// TwinCAT 3 PLC project LabExercise
// ProgramVersion: 3.1.4023.0
// libraries:
//   Tc2_NCI, * (Beckhoff Automation GmbH)
//   Tc2_Standard, * (Beckhoff Automation GmbH)
//   Tc2_System, * (Beckhoff Automation GmbH)
//   Tc3_Module, * (Beckhoff Automation GmbH)
//   VisuDialogs, * (System)
// project tree:
//   Comissioning/Function blocks/ FB_ModifyAutomaticControlSettings.TcPOU (not stored)
//   Comissioning/GVLs/ G_Commissioning.TcGVL (not stored)
//   Comissioning/Struct/ ST_AutomaticControlSettings.TcDUT (not stored), ST_ClosedLoopControlSettings.TcDUT (not stored), ST_MotionReferenceGeneratorSettings.TcDUT (not stored), ST_OpenLoopControlSettings.TcDUT (not stored)
//   ControlBox/Interfaces/ I_ControlBox.TcIO (not stored)
//   ControlBox/Function blocks/ FB_ControlBox.TcPOU, FB_RealControlBox.TcPOU (not stored), FB_VirtualControlBox.TcPOU (not stored)
//   CraneControl/Function blocks/Sub blocks/ FB_ActiveDamping.TcPOU (not stored), FB_Clock.TcPOU (not stored), FB_ClosedLoopControl.TcPOU (not stored), FB_Joystick.TcPOU (not stored), FB_MotionReferenceGenerator_limit.TcPOU (not stored), FB_OpenLoopControl.TcPOU (not stored), FB_ResetIntegralController.TcPOU (not stored), FB_Status.TcPOU (not stored)
//   CraneControl/Enums/ E_Mode.TcDUT (not stored), E_Status.TcDUT (not stored)
//   CraneControl/Function blocks/Main blocks/ FB_AutomaticControl.TcPOU (not stored), FB_ManualControl.TcPOU (not stored)
//   CraneControl/Functions/ F_BarToEng.TcPOU (not stored), F_LminToEng.TcPOU (not stored), F_RadToDeg.TcPOU (not stored)
//   CraneControl/GVLs/ G_Parameters.TcGVL (not stored), G_Work.TcGVL
//   CraneControl/Struct/ ST_ActiveDamping.TcDUT (not stored), ST_Parameters.TcDUT (not stored)
//   / GlobalTextList.TcGTLO (not stored), PlcTask.TcTTO (not stored), Simulator.TcTTO (not stored), Visualization Manager.TcVMO (not stored)
//   HMI/ HMI.TcVIS
//   HMI/Sub/ CommissioningHMI.TcVIS (not stored), VirtualControlBox.TcVIS (not stored)
//   Inputs/ FB_JoystickInputScaling.TcPOU (not stored), FB_PositionInputScaling.TcPOU (not stored), FB_PressureInputScaling.TcPOU (not stored), G_Inputs.TcGVL (not stored), G_Sensors.TcGVL (not stored)
//   Inputs/Struct/ ST_AnalogInput.TcDUT (not stored), ST_AnalogInputStatus.TcDUT (not stored)
//   Internship/ F_PressureSensorInToBar.TcPOU (not stored), V2Q2u.TcPOU
//   Outputs/ FB_ValveOutput.TcPOU (not stored), G_Outputs.TcGVL (not stored)
//   Outputs/Struct/ ST_pValveDeadBand.TcDUT (not stored), ST_ValveOutput.TcDUT (not stored)
//   ControlBox/GVLs/ G_VirtualControlBox.TcGVL (not stored)
//   Programs/ MAIN.TcPOU, P_Commissioning.TcPOU (not stored), P_ControlBox.TcPOU (not stored), P_CraneControl.TcPOU, P_Inputs.TcPOU (not stored), P_OutputNonCompensated.TcPOU, P_Outputs.TcPOU (not stored), P_Simulator.TcPOU (not stored)
//   Simulator/ FB_CraneSimulator.TcPOU, G_Simulator.TcGVL (not stored)
// real-time tasks:
//   TASK PlcTask: cycle T#1ms, priority 20, ADS port 350
//   TASK Simulator: cycle T#100us, priority 1, ADS port 351
// I/O:
//   DEVICE PLC (EtherCAT) (disabled), AmsNetId 10.229.3.117.2.1
//     PLC Rack (EK1200) [EK1200-5000 EtherCAT Power supply (2A E-Bus)]
//       DI (EL1008) [EL1008 8Ch. Dig. Input 24V, 3ms]
//       DO (EL2008) [EL2008 8Ch. Dig. Output 24V, 0.5A]
//       End Cap 4 (EL9011) [EL9011 End Terminal]
//   DEVICE RIO (EtherCAT) (disabled), AmsNetId 10.229.3.117.5.1
//     RIO (EK1100) [EK1100 EtherCAT Coupler (2A E-Bus)]
//       DI (EL1008) [EL1008 8Ch. Dig. Input 24V, 3ms]
//       DO (EL2008) [EL2008 8Ch. Dig. Output 24V, 0.5A]
//       AI1 (EL3068) [EL3068 8Ch. Ana. Input 0-10V]
//       AI2 (EL3068) [EL3068 8Ch. Ana. Input 0-10V]
//       AI3 (EL3174) [EL3174 4Ch. Ana. Input +/-10V Diff., +/-20mA SingleEnded, 16 Bit]
//       AO (EL4104) [EL4104 4Ch. Ana. Output 0-10V, 16bit]
//       End Cap (EL9011) [EL9011 End Terminal]
// variable links:
//   LabExercise/LabExercise Instance <-> PLC (EtherCAT)/PLC Rack (EK1200)/DI (EL1008)
//     PlcTask Inputs/G_Inputs.bTest <-> Channel 1/Input
//   LabExercise/LabExercise Instance <-> PLC (EtherCAT)/PLC Rack (EK1200)/DO (EL2008)
//     PlcTask Outputs/G_Outputs.bTest <-> Channel 1/Output
//   LabExercise/LabExercise Instance <-> RIO (EtherCAT)/RIO (EK1100)/AI1 (EL3068)
//     PlcTask Inputs/G_Inputs.stCylPos.nValue <-> AI Standard Channel 3/Value
//     PlcTask Inputs/G_Inputs.stCylPos.stStatus <-> AI Standard Channel 3/Status
//     PlcTask Inputs/G_Inputs.stJoyX.nValue <-> AI Standard Channel 1/Value
//     PlcTask Inputs/G_Inputs.stJoyX.stStatus <-> AI Standard Channel 1/Status
//     PlcTask Inputs/G_Inputs.stJoyY.nValue <-> AI Standard Channel 2/Value
//     PlcTask Inputs/G_Inputs.stJoyY.stStatus <-> AI Standard Channel 2/Status
//     PlcTask Inputs/G_Inputs.stSpoolPos.nValue <-> AI Standard Channel 4/Value
//     PlcTask Inputs/G_Inputs.stSpoolPos.stStatus <-> AI Standard Channel 4/Status
//   LabExercise/LabExercise Instance <-> RIO (EtherCAT)/RIO (EK1100)/AI2 (EL3068)
//     PlcTask Inputs/G_Inputs.stPressureCompensator.nValue <-> AI Standard Channel 3/Value
//     PlcTask Inputs/G_Inputs.stPressureCompensator.stStatus <-> AI Standard Channel 3/Status
//     PlcTask Inputs/G_Inputs.stPressureLhvSide.nValue <-> AI Standard Channel 5/Value
//     PlcTask Inputs/G_Inputs.stPressureLhvSide.stStatus <-> AI Standard Channel 5/Status
//     PlcTask Inputs/G_Inputs.stPressurePistonSide.nValue <-> AI Standard Channel 4/Value
//     PlcTask Inputs/G_Inputs.stPressurePistonSide.stStatus <-> AI Standard Channel 4/Status
//     PlcTask Inputs/G_Inputs.stPressureReturn.nValue <-> AI Standard Channel 2/Value
//     PlcTask Inputs/G_Inputs.stPressureReturn.stStatus <-> AI Standard Channel 2/Status
//     PlcTask Inputs/G_Inputs.stPressureRodSide.nValue <-> AI Standard Channel 6/Value
//     PlcTask Inputs/G_Inputs.stPressureRodSide.stStatus <-> AI Standard Channel 6/Status
//     PlcTask Inputs/G_Inputs.stPressureSupply.nValue <-> AI Standard Channel 1/Value
//     PlcTask Inputs/G_Inputs.stPressureSupply.stStatus <-> AI Standard Channel 1/Status
//   LabExercise/LabExercise Instance <-> RIO (EtherCAT)/RIO (EK1100)/AI3 (EL3174)
//     PlcTask Inputs/G_Inputs.stFlowReturnSide.nValue <-> AI Standard Channel 1/Value
//     PlcTask Inputs/G_Inputs.stFlowReturnSide.stStatus <-> AI Standard Channel 1/Status
//   LabExercise/LabExercise Instance <-> RIO (EtherCAT)/RIO (EK1100)/AO (EL4104)
//     PlcTask Outputs/G_Outputs.stValveOutput.nValveOutput <-> AO Output Channel 1/Analog output
//   LabExercise/LabExercise Instance <-> RIO (EtherCAT)/RIO (EK1100)/DI (EL1008)
//     PlcTask Inputs/G_Inputs.bAutoModeSelector <-> Channel 1/Input
//     PlcTask Inputs/G_Inputs.bManualModeSelector <-> Channel 2/Input
//     PlcTask Inputs/G_Inputs.bStartButton <-> Channel 3/Input
//     PlcTask Inputs/G_Inputs.bStopButton <-> Channel 4/Input
//   LabExercise/LabExercise Instance <-> RIO (EtherCAT)/RIO (EK1100)/DO (EL2008)
//     PlcTask Outputs/G_Outputs.bGreenLight <-> Channel 1/Output
//     PlcTask Outputs/G_Outputs.bRedLight <-> Channel 2/Output
//     PlcTask Outputs/G_Outputs.stValveOutput.bEnable <-> Channel 3/Output

// ---- CraneControl/GVLs/G_Work.TcGVL
{attribute 'qualified_only'}
VAR_GLOBAL
	eMode 			: E_Mode;
	eStatus 		: E_Status;
	fJoystickY 		: LREAL;
	bFault 			: BOOL;
	bStartButton 	: BOOL;
	bStopButton 	: BOOL;
	fControlOutputNormalized : LREAL;
END_VAR

// ---- ControlBox/Function blocks/FB_ControlBox.TcPOU
FUNCTION_BLOCK FB_ControlBox
VAR_INPUT
	bRealControlBox : BOOL;
	eStatus : E_Status;
END_VAR
VAR_OUTPUT
	eMode : E_Mode;
END_VAR
VAR
	fbVirtualControlBox : FB_VirtualControlBox;
	fbRealControlBox : FB_RealControlBox;
	fbSelectedControlBox : I_ControlBox := fbVirtualControlBox;
END_VAR

IF bRealControlBox THEN
	fbSelectedControlBox := bRealControlBox;
	//fbSelectedControlBox := fbVirtualControlBox;
ELSE
	fbSelectedControlBox := fbVirtualControlBox;
END_IF	
	
fbSelectedControlBox.ModeSelector(
	eMode => eMode
);

fbSelectedControlBox.PushButtons(
	eMode := eMode,
	eStatus := eStatus,
	bStart => G_Work.bStartButton,
	bStop => G_Work.bStopButton 	
);

fbSelectedControlBox.Lamps(
	eMode := eMode,
	eStatus := eStatus
);

fbSelectedControlBox.Joystick(
	eMode := eMode,
	eStatus := eStatus,
	fJoystickY => G_Work.fJoystickY
);

END_FUNCTION_BLOCK

// ---- Internship/V2Q2u.TcPOU
FUNCTION_BLOCK V2Q2u
VAR_INPUT
	Ps	: LREAL;
	Pa	: LREAL;
	Pb	: LREAL;
	y	: LREAL;
END_VAR
VAR_OUTPUT
	u		: LREAL;
	Q_lm	: LREAL;
	dP		: LREAL;
END_VAR
VAR
	phi						: LREAL := 0.7130;
	A						: LREAL := 0.00331;		// Area
	BW 						: LREAL := 0;			// Bandwidth 
	SpoolTravel 			: LREAL := 7.0; 		// Maximum Spool Travel
	dp0						: LREAL := 7E5;			// Pressure drop with compansator 
	fSlopeCharacteristic	: LREAL ;
	dpref					: LREAL ;
	Q						: LREAL ;	
	Q_star					: LREAL ;
	X_dot 					: LREAL ;
END_VAR

fSlopeCharacteristic := (SpoolTravel-BW)/25; 	// Valve Slope Characteristic [mm/(L/min)]  
X_dot := y * 0.1; 

IF X_dot > 0.0 THEN 
    (* '<S1>:1:11' 
	Q := x_dot * A; *)(* Wanted Flow *)
    (* '<S1>:1:12' 
	dP := (Ps-Pa)*1e5; *)
    
    (* '<S1>:1:13'	
	dp_ref := abs(dP_0/dP); *)
     
    (* '<S1>:1:15' 
	Q_star := (Q * sqrt(dp_ref)) * 6e4; *)
	Q := X_dot * A; // Wanted Flow
	dP := (Ps - Pa) * 100000.0;
    dpref := ABS(dP0 / dP); 
	dpref := 1;
	
    Q_star := (Q * SQRT(dpref)) * 60000.0;
    (* Outport: '<Root>/u' *)
    (* Referance Flow [L/min] *)
    (* '<S1>:1:16' 
	u := (Q_star * a + BW)/SpoolTravel; *)
    u := (Q_star * (fSlopeCharacteristic+BW)) / SpoolTravel; // Control Signal [-1, 1]
ELSIF X_dot < 0.0 THEN 
    (* '<S1>:1:18' elseif x_dot < 0 *)
    Q := X_dot * (A*phi);(* Wanted Flow *)
    (* '<S1>:1:20' dP := (Ps-Pb)*1e5; *)
    dP := (Ps - Pb) * 100000.0;
    (* '<S1>:1:21' dp_ref := abs(dP_0/dP); *)
    (* dp_ref := 1; *)
    (* '<S1>:1:23' Q_star := (Q * sqrt(dp_ref)) * 6e4; *)
	dpref := ABS(dP0 / dP);
	dpref := 1;
	Q_star := (Q * SQRT(dpref)) * 60000.0;
    (* Outport: '<Root>/u' *)
    (* Referance Flow [L/min] *)
    (* '<S1>:1:24' u := (Q_star * a - BW)/SpoolTravel; *)
	u := (Q_star * (fSlopeCharacteristic - BW)) / SpoolTravel;
    (* Control Signal [-1, 1] *)
ELSE 
    (* '<S1>:1:26' else *)
    (* '<S1>:1:27' Q_star := 0; *)
    Q_star := 0.0;
    (* '<S1>:1:28' dP := 0; *)
    dP := 0.0;
    (* Outport: '<Root>/u' *)
    (* '<S1>:1:29' u := 0; *)
    u := 0.0;
END_IF;

(* Outport: '<Root>/Q_lm' incorporates:
 *  MATLAB Function: '<Root>/V2Q2u' *)
(* '<S1>:1:32' Q_lm := Q_star; *)
(* Q * 6E4; *)
Q_lm := Q_star;

IF u > 1.0 THEN 
    u := 1.0;
ELSIF u < -1.0 THEN 
   	u := -1.0;
END_IF;

END_FUNCTION_BLOCK

// ---- Programs/MAIN.TcPOU
PROGRAM MAIN
VAR
END_VAR

P_Commissioning();
P_ControlBox();
P_CraneControl();
P_OutputNonCompensated();
P_Inputs();

END_PROGRAM

// ---- Programs/P_CraneControl.TcPOU
PROGRAM P_CraneControl
VAR
 	fbStatus 					: FB_Status;
	fbRunningClock 				: FB_Clock;
	fbManualControl 			: FB_ManualControl; 
	bEnableManualControl 		: BOOL;
	fbAutomaticControl 			: FB_AutomaticControl;
	bEnableAutomaticControl 	: BOOL; 
	fbActiveDamping 			: FB_ActiveDamping;
	fControlOutputNormalized 	: LREAL; 
	
	ADtest0 : LREAL;
	ADtest1 : LREAL;
	ADtest2 : LREAL;
	ADtest : BOOL;
END_VAR

fbStatus(
bFault := G_Work.bFault,
eMode := G_Work.eMode,
fTime := fbRunningClock.fTime,
eStatus => G_Work.eStatus
);

fbRunningClock(
	bStart := (fbStatus.eStatus = E_Status.Starting) OR (fbStatus.eStatus = E_Status.Running),
	bStop := (fbStatus.eStatus = E_Status.Stopping),
	fCycleTime := G_Parameters.stParam.fCyclicTime
);

fbManualControl(
	eMode := G_Work.eMode,
	eStatus := G_Work.eStatus,
	stParam := G_Parameters.stParam, 
);

fbAutomaticControl(
	eMode := G_Work.eMode,
	eStatus := G_Work.eStatus,
	stAutomaticControlSettings := G_Commissioning.stAutomaticControlSettings,
	stMotionReferenceGeneratorSettings := G_Commissioning.stMotionReferenceGeneratorSettings,
	stParam := G_Parameters.stParam,
	fPositionFeedback := G_Sensors.fPistonPosition
);

fbActiveDamping(
	ssMethodType := BOOL_TO_SINT(G_Commissioning.stAutomaticControlSettings.bEnableActiveDamping),
	bEnable := (fbStatus.eStatus = E_Status.Running),
	stParam := G_Parameters.stParam,
	fPressurePistonSide_Pa := F_BarToEng(G_Sensors.fPressurePistonSide),
	fPressureRodSide_Pa := F_BarToEng(G_Sensors.fPressureRodSide)
);

IF (G_Work.eMode = E_Mode.Manual AND G_Work.eStatus = E_Status.Running) THEN
	fControlOutputNormalized := LIMIT(-1.0, (fbManualControl.fControlOutputNormalized - fbActiveDamping.fPressureFeedbackNormalized), 1.0);
ELSIF (G_Work.eMode = E_Mode.Auto AND G_Work.eStatus = E_Status.Running) THEN
	fControlOutputNormalized := LIMIT(-1.0, (-fbAutomaticControl.fControlOutputNormalized - fbActiveDamping.fPressureFeedbackNormalized), 1.0);
ELSE
	fControlOutputNormalized := 0.0;
END_IF

//G_Work.fControlOutputNormalized := fControlOutputNormalized;

END_PROGRAM

// ---- Programs/P_OutputNonCompensated.TcPOU
PROGRAM P_OutputNonCompensated
VAR
	fbValueInput 	: V2Q2u;
END_VAR

fbValueInput(
	Ps 	:= G_Sensors.fPressureSupply,
	Pa 	:= G_Sensors.fPressurePistonSide,
  	//Pa 	:= G_Simulator.fPistonSidePressure,
	Pb 	:= G_Sensors.fPressureRodSide,
  	//Pb 	:= G_Simulator.fRodSidePressure,
	y 	:= G_Sensors.fJoystickY,
	u	=> G_Work.fControlOutputNormalized
);

END_PROGRAM

// ---- Simulator/FB_CraneSimulator.TcPOU
FUNCTION_BLOCK FB_CraneSimulator
VAR_INPUT
	ssMethodType: SINT;
	uDCV: LREAL;
END_VAR
VAR_OUTPUT
	xm: LREAL;
	ppbar: LREAL;
	prbar: LREAL;
END_VAR
VAR
	pLS: LREAL;
	QDCV_out: LREAL;
	rtb_xDot: LREAL;
	rtb_xDotDot: LREAL;
	temp1: LREAL;
	temp2: LREAL;
	temp3: LREAL;
	temp4: LREAL;
	c_DiscreteTimeIntegrator2_D: LREAL;
	c_DiscreteTimeIntegrator3_D: LREAL;
	c_DiscreteTimeIntegrator_DS: LREAL;
	c_DiscreteTimeIntegrator4_D: LREAL;
END_VAR



CASE ssMethodType OF
    0: 
        (* SystemInitialize for Atomic SubSystem: '<Root>/FB_CraneSimulator' *)
        (* InitializeConditions for DiscreteIntegrator: '<S1>/Discrete-Time Integrator' *)
        c_DiscreteTimeIntegrator_DS := 4.377E+6;
        (* InitializeConditions for DiscreteIntegrator: '<S1>/Discrete-Time Integrator2' *)
        c_DiscreteTimeIntegrator2_D := 0.0;
        (* InitializeConditions for DiscreteIntegrator: '<S1>/Discrete-Time Integrator3' *)
        c_DiscreteTimeIntegrator3_D := 0.0;
        (* InitializeConditions for DiscreteIntegrator: '<S1>/Discrete-Time Integrator4' *)
        c_DiscreteTimeIntegrator4_D := 468300.0;
        (* End of SystemInitialize for SubSystem: '<Root>/FB_CraneSimulator' *)
    1: 
        (* Outputs for Atomic SubSystem: '<Root>/FB_CraneSimulator' *)
        (* DiscreteIntegrator: '<S1>/Discrete-Time Integrator2' *)
        rtb_xDot := c_DiscreteTimeIntegrator2_D;
        (* Outport: '<Root>/x [m]' incorporates:
         *  DiscreteIntegrator: '<S1>/Discrete-Time Integrator3' *)
        xm := c_DiscreteTimeIntegrator3_D;
        (* Outport: '<Root>/pp [bar]' incorporates:
         *  DiscreteIntegrator: '<S1>/Discrete-Time Integrator'
         *  Gain: '<S1>/Gain' *)
        ppbar := 1.0E-5 * c_DiscreteTimeIntegrator_DS;
        (* Outport: '<Root>/pr [bar]' incorporates:
         *  DiscreteIntegrator: '<S1>/Discrete-Time Integrator4'
         *  Gain: '<S1>/Gain1' *)
        prbar := 1.0E-5 * c_DiscreteTimeIntegrator4_D;
        (* MATLAB Function: '<S1>/MATLAB Function' incorporates:
         *  DiscreteIntegrator: '<S1>/Discrete-Time Integrator'
         *  DiscreteIntegrator: '<S1>/Discrete-Time Integrator2'
         *  DiscreteIntegrator: '<S1>/Discrete-Time Integrator3'
         *  DiscreteIntegrator: '<S1>/Discrete-Time Integrator4' *)
        (* Parameters *)
        (* MATLAB Function 'FB_CraneSimulator/MATLAB Function': '<S2>:1' *)
        (* '<S2>:1:3' Fexternal = 1.3365e+04; *)
        (* [N] *)
        (* '<S2>:1:4' mEffective = 1.3365e+04; *)
        (* [kg] *)
        (* '<S2>:1:5' kFric = 4000; *)
        (* [N/(ms)] *)
        (* '<S2>:1:6' Apiston = 0.0033; *)
        (* [m^2] *)
        (* '<S2>:1:7' Aannulus = 0.0023; *)
        (* [m^2] *)
        (* '<S2>:1:8' beta = 1.0e9; *)
        (* [Pa] *)
        (* '<S2>:1:9' pSupply = 180e5; *)
        (* [Pa] *)
        (* '<S2>:1:10' pReturn = 1.1e5; *)
        (* [Pa] *)
        (* '<S2>:1:11' MaxStroke = 0.5; *)
        (* [m] *)
        (* '<S2>:1:12' VCyl_A = 1.0e-03; *)
        (* '<S2>:1:13' VCyl_B = 1.25e-03; *)
        (* '<S2>:1:14' p_nom_DCV = 7e5; *)
        (* '<S2>:1:15' Q1_ref_DCV = 20/6e4; *)
        (* '<S2>:1:16' kv1_DCV = Q1_ref_DCV/sqrt(p_nom_DCV); *)
        (* '<S2>:1:17' p0 = 7e5; *)
        (* compensator crack pressure *)
        (* Directional Control Valve - Lifting Cylinder  *)
        (* LS Pressure *)
        (* '<S2>:1:20' if uDCV > 0 *)

        IF uDCV > 0.0 THEN 
            (* '<S2>:1:21' pLS = pPiston; *)
            pLS := c_DiscreteTimeIntegrator_DS;
        ELSIF uDCV < 0.0 THEN 
            (* '<S2>:1:22' elseif uDCV < 0 *)
            (* '<S2>:1:23' pLS = pRod; *)
            pLS := c_DiscreteTimeIntegrator4_D;
        ELSE 
            (* '<S2>:1:24' else *)
            (* '<S2>:1:25' pLS = 0; *)
            pLS := 0.0;
        END_IF;

        (* '<S2>:1:28' if pLS<0 *)

        IF pLS < 0.0 THEN 
            (* '<S2>:1:29' pLS = 0; *)
            pLS := 0.0;
        END_IF;

        (* Pressure Compensator *)
        (* '<S2>:1:33' pPC = 0; *)
        (* '<S2>:1:35' if p0 <= (pSupply - pLS) *)

        IF 700000.0 <= (1.8E+7 - pLS) THEN 
            (* '<S2>:1:36' pPC = pLS+p0; *)
            pLS := pLS + 700000.0;
        ELSE 
            (* '<S2>:1:37' elseif 0 < (pSupply - pLS) < p0 *)
            (* '<S2>:1:38' pPC = pSupply-pLS; *)
            pLS := 1.8E+7 - pLS;
        END_IF;

        (* '<S2>:1:43' if pPC<0 *)

        IF pLS < 0.0 THEN 
            (* '<S2>:1:44' pPC = 0; *)
            pLS := 0.0;
        END_IF;

        (* Orifice Equations *)
        (* '<S2>:1:47' if uDCV > 0 *)

        IF uDCV > 0.0 THEN 
            (* '<S2>:1:48' QDCV_in =  kv1_DCV*uDCV*sign(pPC-pPiston)*sqrt(abs(pPC-pPiston)); *)
            pLS := pLS - c_DiscreteTimeIntegrator_DS;

            IF pLS < 0.0 THEN 
                rtb_xDotDot := -1.0;
            ELSIF pLS > 0.0 THEN 
                rtb_xDotDot := 1.0;
            ELSE 
                rtb_xDotDot := pLS;
            END_IF;

            temp3 := ABS(pLS);
            pLS := ((3.9840953644479785E-7 * uDCV) * rtb_xDotDot) * SQRT(temp3);
            (* '<S2>:1:49' QDCV_out = kv1_DCV*uDCV*sign(pRod-pReturn)*sqrt(abs(pRod-pReturn)); *)

            IF (c_DiscreteTimeIntegrator4_D - 110000.0) < 0.0 THEN 
                rtb_xDotDot := -1.0;
            ELSIF (c_DiscreteTimeIntegrator4_D - 110000.0) > 0.0 THEN 
                rtb_xDotDot := 1.0;
            ELSE 
                rtb_xDotDot := c_DiscreteTimeIntegrator4_D - 110000.0;
            END_IF;

            temp4 := ABS(c_DiscreteTimeIntegrator4_D - 110000.0);
            QDCV_out := ((3.9840953644479785E-7 * uDCV) * rtb_xDotDot) * SQRT(temp4);
        ELSIF uDCV < 0.0 THEN 
            (* '<S2>:1:50' elseif uDCV < 0 *)
            (* '<S2>:1:51' QDCV_out =  kv1_DCV*uDCV*sign(pPC-pRod)*sqrt(abs(pPC-pRod)); *)
            pLS := pLS - c_DiscreteTimeIntegrator4_D;

            IF pLS < 0.0 THEN 
                rtb_xDotDot := -1.0;
            ELSIF pLS > 0.0 THEN 
                rtb_xDotDot := 1.0;
            ELSE 
                rtb_xDotDot := pLS;
            END_IF;

            temp1 := ABS(pLS);
            QDCV_out := ((3.9840953644479785E-7 * uDCV) * rtb_xDotDot) * SQRT(temp1);
            (* '<S2>:1:52' QDCV_in =  kv1_DCV*uDCV*sign(pRod-pReturn)*sqrt(abs(pRod-pReturn)); *)

            IF (c_DiscreteTimeIntegrator4_D - 110000.0) < 0.0 THEN 
                rtb_xDotDot := -1.0;
            ELSIF (c_DiscreteTimeIntegrator4_D - 110000.0) > 0.0 THEN 
                rtb_xDotDot := 1.0;
            ELSE 
                rtb_xDotDot := c_DiscreteTimeIntegrator4_D - 110000.0;
            END_IF;

            temp2 := ABS(c_DiscreteTimeIntegrator4_D - 110000.0);
            pLS := ((3.9840953644479785E-7 * uDCV) * rtb_xDotDot) * SQRT(temp2);
        ELSE 
            (* '<S2>:1:53' else *)
            (* '<S2>:1:54' QDCV_in = 0; *)
            pLS := 0.0;
            (* '<S2>:1:55' QDCV_out = 0; *)
            QDCV_out := 0.0;
        END_IF;

        (* Pressure Gradients *)
        (* '<S2>:1:58' VA = VCyl_A + x*Apiston; *)
        (* '<S2>:1:59' VB =  VCyl_B + (MaxStroke - x)*Aannulus; *)
        (* '<S2>:1:60' VA_dot = Apiston*xDot; *)
        (* '<S2>:1:61' VB_dot = -Aannulus*xDot; *)
        (* '<S2>:1:62' pPistonDot = beta/VA*(QDCV_in - VA_dot); *)
        (* '<S2>:1:63' pRodDot = beta/VB*(-QDCV_out - VB_dot); *)
        QDCV_out := (1.0E+9 / (((0.5 - c_DiscreteTimeIntegrator3_D) * 0.0023) + 0.00125)) * (( -QDCV_out) - (-0.0023 * c_DiscreteTimeIntegrator2_D));
        (* Viscouse Friction *)
        (* '<S2>:1:66' Ffric = kFric*xDot; *)
        (* Hydraulic Force *)
        (* '<S2>:1:69' Fhyd = pPiston*Apiston - pRod*Aannulus; *)
        (* Newton Second Law of Motion *)
        (* '<S2>:1:72' xDotDot = (Fhyd - Ffric - Fexternal)/mEffective; *)
        rtb_xDotDot := ((((c_DiscreteTimeIntegrator_DS * 0.0033) - (c_DiscreteTimeIntegrator4_D * 0.0023)) - (4000.0 * c_DiscreteTimeIntegrator2_D)) - 23365.0) / 23365.0;
        (* Update for DiscreteIntegrator: '<S1>/Discrete-Time Integrator' incorporates:
         *  DiscreteIntegrator: '<S1>/Discrete-Time Integrator2'
         *  DiscreteIntegrator: '<S1>/Discrete-Time Integrator3'
         *  MATLAB Function: '<S1>/MATLAB Function' *)
        c_DiscreteTimeIntegrator_DS := (((1.0E+9 / ((c_DiscreteTimeIntegrator3_D * 0.0033) + 0.001)) * (pLS - (0.0033 * c_DiscreteTimeIntegrator2_D))) * 0.0001) + c_DiscreteTimeIntegrator_DS;

        IF c_DiscreteTimeIntegrator_DS >= 1.8E+7 THEN 
            c_DiscreteTimeIntegrator_DS := 1.8E+7;
        ELSIF c_DiscreteTimeIntegrator_DS <= 110000.0 THEN 
            c_DiscreteTimeIntegrator_DS := 110000.0;
        END_IF;

        (* End of Update for DiscreteIntegrator: '<S1>/Discrete-Time Integrator' *)
        

        (* Update for DiscreteIntegrator: '<S1>/Discrete-Time Integrator2' *)
        c_DiscreteTimeIntegrator2_D := (0.0001 * rtb_xDotDot) + c_DiscreteTimeIntegrator2_D;

        IF c_DiscreteTimeIntegrator2_D >= 0.12 THEN 
            c_DiscreteTimeIntegrator2_D := 0.12;
        ELSIF c_DiscreteTimeIntegrator2_D <= -0.12 THEN 
            c_DiscreteTimeIntegrator2_D := -0.12;
        END_IF;

        (* End of Update for DiscreteIntegrator: '<S1>/Discrete-Time Integrator2' *)
        

        (* Update for DiscreteIntegrator: '<S1>/Discrete-Time Integrator3' *)
        c_DiscreteTimeIntegrator3_D := (0.0001 * rtb_xDot) + c_DiscreteTimeIntegrator3_D;

        IF c_DiscreteTimeIntegrator3_D >= 0.5 THEN 
            c_DiscreteTimeIntegrator3_D := 0.5;
        ELSIF c_DiscreteTimeIntegrator3_D <= 0.0 THEN 
            c_DiscreteTimeIntegrator3_D := 0.0;
        END_IF;

        (* End of Update for DiscreteIntegrator: '<S1>/Discrete-Time Integrator3' *)
        

        (* Update for DiscreteIntegrator: '<S1>/Discrete-Time Integrator4' *)
        c_DiscreteTimeIntegrator4_D := (0.0001 * QDCV_out) + c_DiscreteTimeIntegrator4_D;

        IF c_DiscreteTimeIntegrator4_D >= 1.8E+7 THEN 
            c_DiscreteTimeIntegrator4_D := 1.8E+7;
        ELSIF c_DiscreteTimeIntegrator4_D <= 110000.0 THEN 
            c_DiscreteTimeIntegrator4_D := 110000.0;
        END_IF;

        (* End of Update for DiscreteIntegrator: '<S1>/Discrete-Time Integrator4' *)
        (* End of Outputs for SubSystem: '<Root>/FB_CraneSimulator' *)
END_CASE;

END_FUNCTION_BLOCK

// ---- HMI/HMI.TcVIS
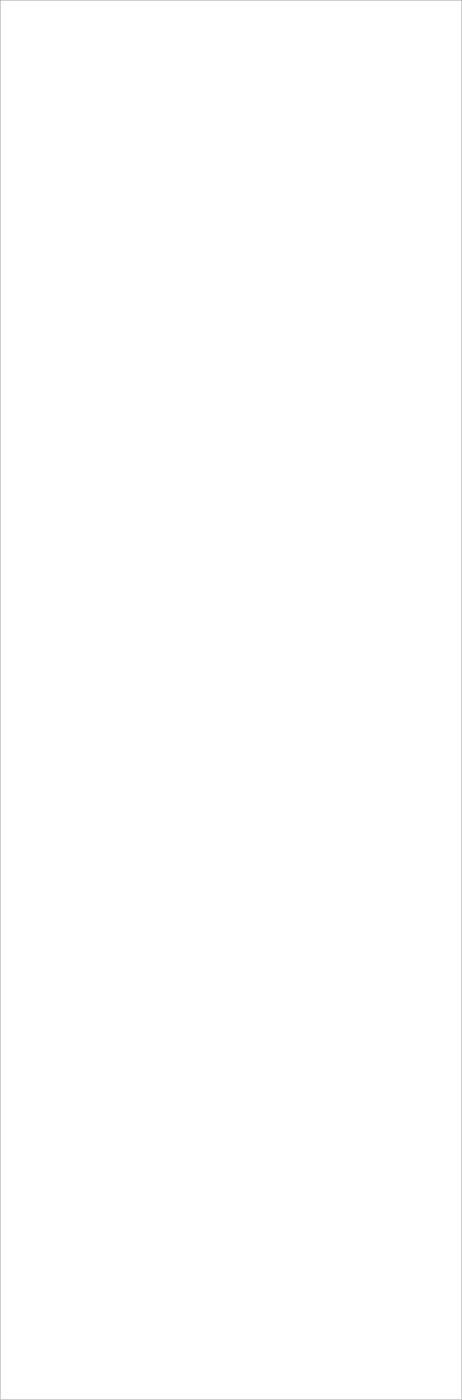
VISUALIZATION HMI  // 1197x3621
    TabControl (4,-3621 1193x643)
        shows VirtualControlBox()
        shows CommissioningHMI()
        [0]: TabTitle=ControlBox
        [1]: TabTitle=Comissioning
END_VISUALIZATION
